{attribute addProperty BoxType "EPP2339-0003-0016"}
{attribute addProperty Id "InputAT %I*ARRAY[0 ..7] OF BOOL6480Sync_errorAT %I*BOOL8114TxPDO_StateAT %I*BOOL8115TxPDO_ToggleAT %I*BOOL8116"}
{attribute addProperty CRC "285397209"}
{attribute addProperty SizeInBites "88"}
{attribute addProperty SizeInBytes "11"}
TYPE DI_Inputs_Channel_595007DD :
STRUCT
	{attribute addProperty Name "Input"}
	Input AT %I* : ARRAY[0 ..7] OF BOOL;
	{attribute addProperty Name "Sync_error"}
	Sync_error AT %I* : BOOL;
	{attribute addProperty Name "TxPDO_State"}
	TxPDO_State AT %I* : BOOL;
	{attribute addProperty Name "TxPDO_Toggle"}
	TxPDO_Toggle AT %I* : BOOL;
END_STRUCT
END_TYPE

(* stored: Version 1.2.0.0, ProductVersion 3.1.4024.9
   DUT DI_Inputs_Channel_595007DD: Id {732b988b-73c1-4d59-bcd5-1ac60e912809} *)
